(* CoDeSys 2.3 library: EQ_GT.lib *)
(* Libraries: STANDARD.LIB 5.6.98 11:03:02 *)

(* POU MAIN, LD *)
PROGRAM MAIN
VAR
END_VAR
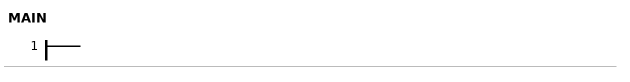
_LD_ (* Ladder Diagram *)
NETWORK 1
	*
_END_LD_
(* the same logic as Structured Text *)
(* Network 1 *)
END_PROGRAM

(* POU EQ_GT, LD *)
FUNCTION_BLOCK EQ_GT
VAR_INPUT
	INT_SOURCE_A: INT;
	INT_SOURCE_B: INT;
END_VAR
VAR_OUTPUT
	SIGNAL_BOOL: BOOL;
END_VAR
VAR
	M0: BOOL;
	M1: BOOL;
END_VAR
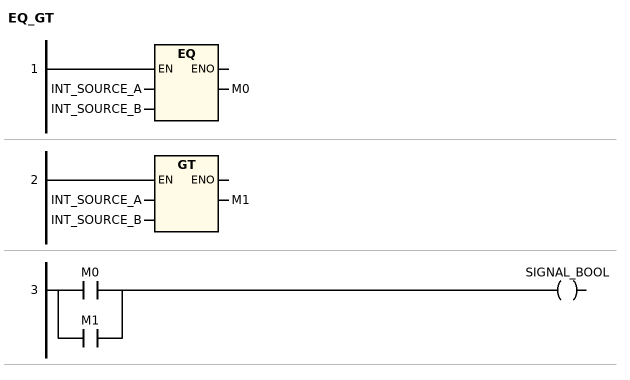
_LD_ (* Ladder Diagram *)
NETWORK 1
	*
		EN --- EQ(INT_SOURCE_A, INT_SOURCE_B) => M0
NETWORK 2
	*
		EN --- GT(INT_SOURCE_A, INT_SOURCE_B) => M1
NETWORK 3
	{ [M0] | [M1] } --- (SIGNAL_BOOL)
_END_LD_
(* the same logic as Structured Text *)
(* Network 1 *)
M0 := INT_SOURCE_A = INT_SOURCE_B;
(* Network 2 *)
M1 := INT_SOURCE_A > INT_SOURCE_B;
(* Network 3 *)
SIGNAL_BOOL := M0 OR M1;
END_FUNCTION_BLOCK
